FUNCTION_BLOCK FB_mbWriteSingleReg
VAR_INPUT
	bExecute : BOOL;
	Robot : STRING;
	Register : WORD;
	Value : WORD;
END_VAR
VAR_OUTPUT
	bBusy : BOOL;
END_VAR
VAR
	mbWrite : FB_mbWriteRegs;
	state : int;
END_VAR

(* 
FB_mbWriteSingleReg - Function Block that can be called to write a single MODBUS register
	INPUTS:
		- Robot: 'UR5' or 'UR3'
		- Register: register number to write
		- Value: value to write
	OUTPUTS
		
*)

IF bExecute THEN
	// Set/Determine State of Function block
	CASE state OF
		0:
			// Set function block vairables
			mbWrite.nQuantity := 1;
			mbWrite.cbLength := 2;
			
			IF Robot='UR5' THEN
				mbWrite.sIPAddr := Global.stUR5.IP;
				mbWrite.nTCPPort := Global.stUR5.mbPort;
				mbWrite.nUnitID := Global.stUR5.unitID;
			ELSIF Robot='UR3' THEN
				mbWrite.sIPAddr := Global.stUR3.IP;
				mbWrite.nTCPPort := Global.stUR3.mbPort;
				mbWrite.nUnitID := Global.stUR3.unitID;
			END_IF
			
			mbWrite.pSrcAddr := ADR(Value);
			mbWrite.nMBAddr := Register;
			mbWrite.bExecute := TRUE;
			
			// Set fuctionblock busy bit
			bBusy := TRUE;
			
			state := 10;
	
		10:
			IF NOT mbWrite.bBusy THEN
				mbWrite.bExecute :=FALSE;
				state := 0;
			END_IF
	END_CASE
	
	// Run function block
	mbWrite();
END_IF

END_FUNCTION_BLOCK

(* stored: Version 1.1.0.1, ProductVersion 3.1.4020.12
   POU FB_mbWriteSingleReg: Id {0feda740-7134-4840-abdb-d6e810a3aa80}, SpecialFunc None *)
